// TwinCAT 3 PLC project Untitled1
// ProgramVersion: 3.1.4024.12
// libraries:
//   Tc2_MC2, * (Beckhoff Automation GmbH)
//   Tc2_Standard, * (Beckhoff Automation GmbH)
//   Tc2_System, * (Beckhoff Automation GmbH)
//   Tc3_Module, * (Beckhoff Automation GmbH)
// project tree:
//   GVLs/ GVL.TcGVL
//   / PlcTask.TcTTO
//   POUs/01_SubModules/Axis/ FB_Axis.TcPOU, FB_AxisPTP.TcPOU
//   POUs/ MAIN.TcPOU
// real-time tasks:
//   TASK PlcTask: cycle T#10ms, priority 20, ADS port 350
// motion (NC):
//   TASK NC-Task 1 SAF: cycle T#2ms, priority 4, ADS port 501
//   TASK NC-Task 1 SVB: cycle T#10ms, priority 8, ADS port 511
//   AXIS Axis 1 (id 1)
//     Dynamic: Acceleration=5908.72576, Deceleration=5908.72576, Jerk=17726.17728
//     Velo: RefSearch=39.3915050666667, RefSync=39.3915050666667, SlowManual=196.957525333333, FastManual=1181.745152, Fast=3939.15050666667, Maximum=3939.15050666667
//     OtherSettings: AllowMotionCmdToSlave=true
//     encoder EncType=19
//       EncPara: ScaleFactorNumerator=104.8576, ScaleFactorDenominator=1048576, MaxCount=#xffffffff
//     drive DrvType=16
//       DrvPara: MaxCount=#xffffffff, DriveControlDWord=#x00020000
//         Analog: VeloReferenz=4333.06555733333, VeloScale=32, TorqueSetpointScale=10, ScaleFactorActTorque=0.1
//         TimeComp: TaskDelayCycles=1
//     controller CtrType=1
//       CtrPara: PriorControlFactor=1
//         PosDiffControl: Range=40
//         Observer: BandWidth=20
//   AXIS Axis 2 (id 2)
//     Dynamic: Acceleration=15295.0528, Deceleration=15295.0528, Jerk=45885.1584
//     Velo: RefSearch=101.967018666667, RefSync=101.967018666667, SlowManual=509.835093333333, FastManual=3059.01056, Fast=10196.7018666667, Maximum=10196.7018666667
//     OtherSettings: AllowMotionCmdToSlave=true
//     encoder EncType=8
//       EncPara: ScaleFactorNumerator=104.8576, ScaleFactorDenominator=1048576, MaxCount=#xffffffff
//     drive DrvType=9
//       DrvPara: MaxCount=#xffffffff, DriveControlDWord=#x00030100
//         Analog: VeloReferenz=11216.3720533333, VeloScale=1.02400649589962, TorqueSetpointScale=10, ScaleFactorActTorque=0.1
//         TimeComp: TaskDelayCycles=1
//     controller CtrType=1
//       CtrPara: PriorControlFactor=1
//         Observer: BandWidth=20
//   AXIS Axis 3 (id 3)
//     Dynamic: Acceleration=15587.2, Deceleration=15587.2, Jerk=46761.7
//     Velo: RefSearch=103.9149824, RefSync=103.9149824, SlowManual=519.574912, FastManual=3117.449472, Fast=10391.49824, Maximum=10391.5
//     OtherSettings: AllowMotionCmdToSlave=true
//     encoder EncType=8
//       EncPara: ScaleFactorNumerator=104.8576, ScaleFactorDenominator=1048576, MaxCount=#xffffffff
//     drive DrvType=9
//       DrvPara: MaxCount=#xffffffff, DriveControlDWord=#x00030100
//         Analog: VeloReferenz=11430.648064, VeloScale=1.02400649589962, TorqueSetpointScale=10, ScaleFactorActTorque=0.1
//         TimeComp: TaskDelayCycles=1
//     controller CtrType=1
//       CtrPara: PriorControlFactor=1
//         Observer: BandWidth=20
// I/O:
//   DEVICE Device 1 (EtherCAT), AmsNetId 5.79.65.80.2.1
//     Term 1 (EK1200) [EK1200-5000 EtherCAT Power supply (2A E-Bus)]
//       Term 2 (EL1819) [EL1819 16Ch. Dig. Input 24V, 10µs]
//       Term 3 (EL2809) [EL2809 16Ch. Dig. Output 24V, 0.5A]
//       Term 4 (EL3064) [EL3064 4Ch. Ana. Input 0-10V]
//       Term 5 (EL4004) [EL4004 4Ch. Ana. Output 0-10V, 12bit]
//       Term 6 (EL7201) [EL7201 1Ch. MDP742 Servo motor output stage (50V, 4A)]
//       Term 7 (EL9510) [EL9510 Power supply terminal 10V]
//       Term 8 (EL9011) [EL9011 End Terminal]
//   DEVICE Device 4 (EtherCAT), AmsNetId 5.79.65.80.5.1
//     Drive 9 (AX5203-0000-0203) [AX5203-0000-0203 EtherCAT Drive (SoE, 2 Ch.)]
//     Term 10 (EK1100) [EK1100 EtherCAT Coupler (2A E-Bus)]
//       Term 11 (EL6900) [EL6900, TwinSAFE PLC]
//       Term 12 (EL1904) [EL1904, 4 Ch. Safety Input 24V, TwinSAFE]
//         modules: Module 1 (FSOES)
//       Term 13 (EL1904) [EL1904, 4 Ch. Safety Input 24V, TwinSAFE]
//         modules: Module 1 (FSOES)
//       Term 14 (EL2904) [EL2904, 4 Ch. Safety Output 24V, 0.5A, TwinSAFE]
//         modules: Module 1 (FSOES), Module 2 (DO)
//       Term 7 (EL9011) [EL9011 End Terminal]
// variable links:
//   Device 4 (EtherCAT) <-> Device 4 (EtherCAT)/Term 10 (EK1100)/Term 11 (EL6900)
//     Term 10 (EK1100)/Term 12 (EL1904)/Module 1 (FSOES)/TxPDO/FSOE <-> ConnectionOutputs/Message_5 RxPDO
//   Device 4 (EtherCAT) <-> Device 4 (EtherCAT)/Term 10 (EK1100)/Term 12 (EL1904)
//     Term 10 (EK1100)/Term 11 (EL6900)/ConnectionInputs/Message_5 TxPDO <-> Module 1 (FSOES)/RxPDO/FSOE
//   Device 4 (EtherCAT) <-> Device 4 (EtherCAT)/Term 10 (EK1100)/Term 14 (EL2904)
//     Term 10 (EK1100)/Term 11 (EL6900)/ConnectionInputs/Message_6 TxPDO <-> Module 1 (FSOES)/RxPDO/FSOE
//     Term 10 (EK1100)/Term 11 (EL6900)/ConnectionOutputs/Message_6 RxPDO <-> Module 1 (FSOES)/TxPDO/FSOE
//   NC-Task 1 SAF/Axes/Axis 1 <-> Device 1 (EtherCAT)/Term 1 (EK1200)/Term 6 (EL7201)
//     Drive/Inputs/In/nDcOutputTime <-> InfoData/DcOutputShift
//     Drive/Inputs/In/nState1 <-> DRV Statusword/Statusword
//     Drive/Inputs/In/nState2 <-> DRV Statusword/Statusword @bit 8
//     Drive/Inputs/In/nState4 @bit 1 <-> WcState/InputToggle
//     Drive/Inputs/In/nState4 <-> WcState/WcState
//     Drive/Outputs/Out/nCtrl1 <-> DRV Controlword/Controlword
//     Drive/Outputs/Out/nCtrl2 <-> DRV Controlword/Controlword @bit 8
//     Drive/Outputs/Out/nDataOut2 <-> DRV Target velocity/Target velocity
//     Enc/Inputs/In/nDataIn1 <-> FB Position/Position
//     Enc/Inputs/In/nDcInputTime <-> InfoData/DcInputShift
//     Enc/Inputs/In/nState4 @bit 1 <-> WcState/InputToggle
//     Enc/Inputs/In/nState4 <-> WcState/WcState
//   NC-Task 1 SAF/Axes/Axis 2 <-> Device 4 (EtherCAT)/Drive 9 (AX5203-0000-0203)
//     Drive/Inputs/In/nDataIn1 <-> AT 1/Following distance
//     Drive/Inputs/In/nDcOutputTime <-> InfoData/DcOutputShift
//     Drive/Inputs/In/nState1 <-> AT 1/Drive status word @bit 8
//     Drive/Inputs/In/nState2 <-> AT 1/Drive status word
//     Drive/Inputs/In/nState4 @bit 1 <-> WcState/InputToggle
//     Drive/Inputs/In/nState4 <-> WcState/WcState
//     Drive/Outputs/Out/nCtrl1 <-> MDT 1/Master control word @bit 8
//     Drive/Outputs/Out/nDataOut1 <-> MDT 1/Position command value
//     Enc/Inputs/In/nDataIn1 <-> AT 1/Position feedback 1 value
//     Enc/Inputs/In/nDcInputTime <-> InfoData/DcInputShift
//     Enc/Inputs/In/nState4 @bit 1 <-> WcState/InputToggle
//     Enc/Inputs/In/nState4 <-> WcState/WcState
//   NC-Task 1 SAF/Axes/Axis 3 <-> Device 4 (EtherCAT)/Drive 9 (AX5203-0000-0203)
//     Drive/Inputs/In/nDataIn1 <-> AT 2/Following distance
//     Drive/Inputs/In/nDcOutputTime <-> InfoData/DcOutputShift
//     Drive/Inputs/In/nState1 <-> AT 2/Drive status word @bit 8
//     Drive/Inputs/In/nState2 <-> AT 2/Drive status word
//     Drive/Inputs/In/nState4 @bit 1 <-> WcState/InputToggle
//     Drive/Inputs/In/nState4 <-> WcState/WcState
//     Drive/Outputs/Out/nCtrl1 <-> MDT 2/Master control word @bit 8
//     Drive/Outputs/Out/nDataOut1 <-> MDT 2/Position command value
//     Enc/Inputs/In/nDataIn1 <-> AT 2/Position feedback 1 value
//     Enc/Inputs/In/nDcInputTime <-> InfoData/DcInputShift
//     Enc/Inputs/In/nState4 @bit 1 <-> WcState/InputToggle
//     Enc/Inputs/In/nState4 <-> WcState/WcState
//   Untitled1/Untitled1 Instance <-> Device 1 (EtherCAT)/Term 1 (EK1200)/Term 2 (EL1819)
//     PlcTask Inputs/MAIN.bDigitalInput[1] <-> Channel 1/Input
//     PlcTask Inputs/MAIN.bDigitalInput[2] <-> Channel 2/Input
//     PlcTask Inputs/MAIN.bDigitalInput[3] <-> Channel 3/Input
//   Untitled1/Untitled1 Instance <-> Device 1 (EtherCAT)/Term 1 (EK1200)/Term 4 (EL3064)
//     PlcTask Inputs/MAIN.nAnalogInput <-> AI Standard Channel 1/Value
//   Untitled1/Untitled1 Instance <-> Device 4 (EtherCAT)/Term 10 (EK1100)/Term 11 (EL6900)
//     PlcTask Inputs/GVL.bSafetyComErr <-> StandardInputs/Standard Out Var 4
//     PlcTask Inputs/GVL.bSafetyFbErr <-> StandardInputs/Standard Out Var 3
//     PlcTask Inputs/GVL.bSafetyOutput <-> StandardInputs/Standard Out Var 7
//     PlcTask Outputs/GVL.bSafetyErrorAck <-> StandardOutputs/Standard In Var 1
//     PlcTask Outputs/GVL.bSafetyRun <-> StandardOutputs/Standard In Var 2
//   Untitled1/Untitled1 Instance <-> NC-Task 1 SAF/Axes/Axis 1
//     PlcTask Inputs/MAIN.fbAxis[1].Axis.NcToPlc <-> Outputs/ToPlc
//     PlcTask Outputs/MAIN.fbAxis[1].Axis.PlcToNc <-> Inputs/FromPlc
//   Untitled1/Untitled1 Instance <-> NC-Task 1 SAF/Axes/Axis 2
//     PlcTask Inputs/MAIN.fbAxis[2].Axis.NcToPlc <-> Outputs/ToPlc
//     PlcTask Outputs/MAIN.fbAxis[2].Axis.PlcToNc <-> Inputs/FromPlc
//   Untitled1/Untitled1 Instance <-> NC-Task 1 SAF/Axes/Axis 3
//     PlcTask Inputs/MAIN.fbAxis[3].Axis.NcToPlc <-> Outputs/ToPlc
//     PlcTask Outputs/MAIN.fbAxis[3].Axis.PlcToNc <-> Inputs/FromPlc

CONFIGURATION Untitled1
    RESOURCE PLC ON TwinCAT3
        TASK PlcTask(INTERVAL := T#10ms, PRIORITY := 20);
        PROGRAM MAIN WITH PlcTask : MAIN;
    END_RESOURCE
END_CONFIGURATION

// ---- GVLs/GVL.TcGVL
VAR_GLOBAL
	bSafetyRun AT %Q*		:	BOOL;
	bSafetyErrorAck AT %Q*	:	BOOL;
	bSafetyComErr AT %I*	:	BOOL;
	bSafetyFbErr AT %I*		:	BOOL;
	bSafetyOutput AT %I*	:	BOOL;
END_VAR

// ---- POUs/MAIN.TcPOU
PROGRAM MAIN
VAR
	fbAxis					: ARRAY[1..3] OF FB_AxisPTP;
	nAnalogInput AT %I*		: INT;
	bDigitalInput AT %I*	: ARRAY[1..3] OF BOOL;
	
	eState					: (INIT, READY, RUN);
	fVelocity				: LREAL;
	bRun					: BOOL;
	i						: INT;
END_VAR

fVelocity := INT_TO_LREAL(nAnalogInput) / 32767 * 2000;

FOR i := 1 TO 3 DO
	bRun := bDigitalInput[i];
	CASE eState OF
		INIT:
			fbAxis[i].M_Invoke(FALSE);
		READY:
			fbAxis[i].M_Invoke(TRUE);
		RUN:
			fbAxis[i].fVelocity := fVelocity;
			fbAxis[i].M_MoveFw(bRun);
			fbAxis[i].M_Halt(NOT bRun);
	END_CASE
END_FOR

END_PROGRAM

// ---- POUs/01_SubModules/Axis/FB_AxisPTP.TcPOU
FUNCTION_BLOCK FB_AxisPTP EXTENDS FB_Axis
VAR_INPUT
END_VAR
VAR_OUTPUT
END_VAR
VAR
	// ================== Axis function block =================
	fbMcMove	: MC_MoveVelocity;
	fbMcHalt	: MC_Halt;
	fbMcMovePos	: MC_MoveAbsolute;
	
	// ================== Trigger ==============================
	rTrigHalt		: R_TRIG;
	rTrigMove		: R_TRIG;
	rTrigMovePos	: R_TRIG;
END_VAR

METHOD PUBLIC  M_Halt : BOOL
VAR_INPUT
	bExecute	:	BOOL;
END_VAR
IF NOT bExecute THEN
	bHaltDone := FALSE;
ELSE
	fbMcMove(	Axis	:= Axis,
				Execute := FALSE);
END_IF

rTrigHalt(CLK := bExecute);

IF rTrigHalt.Q THEN
	fbMcHalt(	Axis	:= Axis,
				Execute	:= TRUE);
ELSE
	fbMcHalt(	Axis	:= Axis);
END_IF

IF fbMcHalt.Done OR fbMcHalt.Error OR fbMcHalt.CommandAborted THEN
	bError		:= fbMcHalt.Error;
	nErrorID	:= fbMcHalt.ErrorID;
	bHaltDone	:= fbMcHalt.Done;
	
	fbMcHalt(	Axis	:= Axis,
				Execute	:= FALSE);
END_IF
END_METHOD

METHOD M_MoveFw : BOOL
VAR_INPUT
	bExecute	: BOOL;
END_VAR
IF _fVelocity <= 0 THEN
	bExecute := FALSE;
END_IF

IF bExecute THEN
	fbMcMovePos(Axis := Axis, Execute := FALSE);
ELSE
	;
END_IF

rTrigMove(CLK := bExecute);

IF rTrigMove.Q THEN
	fbMcMove(	Axis		:= Axis,
				Execute		:= TRUE,
				Velocity	:= _fVelocity,
				Direction	:= MC_Positive_Direction);
END_IF

// Error, Command aborted
IF fbMcMove.Error OR fbMcMove.CommandAborted THEN
	bError		:= fbMcMove.Error;
	nErrorID	:= fbMcMove.ErrorID;
	
	fbMcMove(	Axis	:= Axis,
				Execute	:= FALSE);
END_IF
END_METHOD

METHOD PUBLIC M_MovePos : BOOL
VAR_INPUT
	bExecute	: BOOL;
END_VAR
IF _fVelocity <= 0 THEN
	bExecute := FALSE;
END_IF

IF bExecute THEN
	fbMcMove(Axis := Axis, Execute := FALSE);
ELSE
	bMovePosDone := FALSE;
END_IF

rTrigMovePos(CLK := bExecute);

IF rTrigMovePos.Q THEN
	fbMcMovePos(	Axis		:= Axis,
					Execute		:= TRUE,
					Position	:= _fPosition,
					Velocity	:= _fVelocity);
ELSE
	fbMcMovePos(	Axis		:= Axis);
END_IF
		
IF fbMcMovePos.Done OR fbMcMovePos.CommandAborted OR fbMcMovePos.Error THEN
	bMovePosDone	:= fbMcMovePos.Done;
	bError			:= fbMcMovePos.Error;
	nErrorID		:= fbMcMovePos.ErrorID;
	
	fbMcMovePos(Axis := Axis, Execute := FALSE);
END_IF
END_METHOD

METHOD M_Reset : BOOL
VAR_INPUT
	bExecute	: BOOL;
END_VAR
SUPER^.M_Reset(bExecute := bExecute);

IF bExecute THEN
	fbMcMove(	Axis := Axis,
			Execute := FALSE);

	fbMcHalt(	Axis := Axis,
				Execute := FALSE);
END_IF
END_METHOD

END_FUNCTION_BLOCK

// ---- POUs/01_SubModules/Axis/FB_Axis.TcPOU
FUNCTION_BLOCK PUBLIC ABSTRACT FB_Axis
VAR_INPUT
END_VAR
VAR_OUTPUT
	// ================== Axis reference ========================
	Axis				: AXIS_REF;
	
	// ================== State variables =======================
	bError				: BOOL;
	nErrorID			: UDINT;
	bMoves				: BOOL;
	bHaltDone			: BOOL;
	bResetDone			: BOOL;
	bEnableDone			: BOOL;
	bMovePosDone		: BOOL;
END_VAR
VAR
	// ================== Axis function block ===================
	fbMCPower			: MC_Power;
	fbMcReset			: MC_Reset;
	
	// ================== Trigger ================================
	rTrigReset			: R_TRIG;
	
	// ================== Target ================================
	_fVelocity	: LREAL;
	_fPosition	: LREAL;
END_VAR

PROPERTY fPosition : LREAL
GET
fPosition := _fPosition;
END_GET
SET
_fPosition := fPosition;
END_SET
END_PROPERTY

PROPERTY fVelocity : LREAL
GET
fVelocity := _fVelocity;
END_GET
SET
_fVelocity := fVelocity;
END_SET
END_PROPERTY

METHOD PUBLIC ABSTRACT M_Halt : BOOL
VAR_INPUT
	bExecute	:	BOOL;
END_VAR
END_METHOD

METHOD M_Invoke : BOOL
VAR_INPUT
	bEnable		: BOOL;
END_VAR
// ============================================

fbMCPower(	Axis			:= Axis,
			Enable			:= bEnable,
			Enable_Positive	:= bEnable,
			Enable_Negative := bEnable,
			Status			=> bEnableDone);

IF fbMCPower.Error OR Axis.Status.Error THEN
	bError 				:= TRUE;
	nErrorID			:= fbMCPower.ErrorID;
END_IF

Axis.ReadStatus();

bMoves := Axis.Status.Moving;

// ============================================
END_METHOD

METHOD PUBLIC ABSTRACT M_MovePos : BOOL
VAR_INPUT
	bExecute	: BOOL;
END_VAR
END_METHOD

METHOD M_Reset : BOOL
VAR_INPUT
	bExecute	: BOOL;
END_VAR
IF NOT bExecute THEN
	bResetDone		:= FALSE;	
END_IF

rTrigReset(CLK := bExecute);

IF rTrigReset.Q THEN
	bHaltDone		:= FALSE;
	fbMcReset(	Axis	:= Axis,
				Execute	:= TRUE);
ELSE
	fbMcReset(	Axis	:= Axis);
END_IF

// Done / Error
IF fbMcReset.Done OR fbMcReset.Error THEN
	bError			:= fbMcReset.Error;
	nErrorID		:= fbMcReset.ErrorID;
	bResetDone		:= fbMcReset.Done;
	
	fbMcReset(	Axis 	:= Axis,
				Execute	:= FALSE);
END_IF
END_METHOD

END_FUNCTION_BLOCK
